// Interface for a ouble ended queue - Dequeu
INTERFACE I_Deque EXTENDS I_Collection

(* Get item at the back of the deque without removing it. *)
METHOD Back : I_Deque
VAR_INPUT
	Item 	: ANY; (* Variable to store returned item value *)
END_VAR
VAR_OUTPUT
	bSuccess : BOOL;
END_VAR
END_METHOD

(* Gets and remove item at the front of the deque *)
METHOD Dequeue_At_Back : I_Deque
VAR_INPUT
	Item : ANY; (* Variable to store returned item value *)
END_VAR
VAR_OUTPUT
	bSuccess : BOOL;
END_VAR
END_METHOD

(* Gets and remove item at the front of the deque *)
METHOD Dequeue_At_Front : I_Deque
VAR_INPUT
	Item : ANY; (* Variable to store returned item value *)
END_VAR
VAR_OUTPUT
	bSuccess : BOOL;
END_VAR
END_METHOD

(* Removes item at the back of the deque without returning anything *)
METHOD Dequeue_Void_At_Back : I_Deque
VAR_OUTPUT
	bSuccess : BOOL;
END_VAR
END_METHOD

(* Removes item at the front of the deque without returning anything *)
METHOD Dequeue_Void_At_Front : I_Deque
VAR_OUTPUT
	bSuccess : BOOL;
END_VAR
END_METHOD

(* Adds item at the back of the deque *)
METHOD Enqueue_At_Back : I_Deque
VAR_INPUT
	Item : ANY; (* Variable containg data to store on the queue *)
END_VAR
VAR_OUTPUT
	bSuccess : BOOL;
END_VAR
END_METHOD

(* Adds item at the front of the deque *)
METHOD Enqueue_At_Front : I_Deque
VAR_INPUT
	Item : ANY; (* Variable containg data to store on the queue *)
END_VAR
VAR_OUTPUT
	bSuccess : BOOL;
END_VAR
END_METHOD

(* Get item at the front of the deque without removing it. *)
METHOD Front : I_Deque
VAR_INPUT
	Item 	: ANY; (* Variable to store returned item value *)
END_VAR
VAR_OUTPUT
	bSuccess : BOOL;
END_VAR
END_METHOD

(* Get item from the deque without removing it. *)
METHOD Peek : I_Deque
VAR_INPUT
	Item 	: ANY; (* Variable to store returned item value *)
	nIndex 	: DINT; (* Location of item*)
END_VAR
VAR_OUTPUT
	bSuccess : BOOL;
END_VAR
END_METHOD

(* Reverses the order of items in the deque *)
METHOD Reverse : I_Deque
VAR_OUTPUT
	bSuccess : BOOL;
END_VAR
END_METHOD

END_INTERFACE

(* stored: Version 1.1.0.1, ProductVersion 3.1.4024.4
   Itf I_Deque: Id {b4de62e7-c9bc-4fc7-adb1-52b52a474183}
   Method Back: Id {8b450b3e-8ec4-4ad9-9f47-59e1579576f4}
   Method Dequeue_At_Back: Id {5b8dd079-6a6f-427d-99ae-a870b53cadc5}
   Method Dequeue_At_Front: Id {0e319de5-7197-438f-861a-10c203fd3d5e}
   Method Dequeue_Void_At_Back: Id {cbb006e0-82cc-47cd-a8e4-073062834252}
   Method Dequeue_Void_At_Front: Id {ca736cc6-409b-46ad-a6d6-0cddfc4277c5}
   Method Enqueue_At_Back: Id {62a867f5-481a-42d3-a36b-8cc238a4cc06}
   Method Enqueue_At_Front: Id {14d591f4-cc9a-4d06-b446-644046d0139e}
   Method Front: Id {b4f7deb1-4071-4084-97c6-bfb874541217}
   Method Peek: Id {77f94c0d-25bc-4e70-9b68-16157b0ee21a}
   Method Reverse: Id {1acbbe45-3368-408f-9941-1ea4395145d1} *)
